PROGRAM general
VAR PERSISTENT
	//System date time function block
	system_date_time : date_time;
	//Daily reset bit, used throughout the program for any resets
	daily_reset : BOOL;
	//Alarm Acknoweldge unlatch timer
	alarm_ack_ton : ton;
	//Alarm Reset unlatch timer
	alarm_reset_ton : ton;
	//Alarm Ack and reset unlatch timer setpoint
	alarm_ack_unlatch_sp : TIME :=T#1S;
	
	//Always off bit
	always_off : BOOL := FALSE;
	
	//PLC States - move as needed
	ed_routine_idle : BOOL;
	ed_routine_cip : BOOL;
	ed_routine_manual : BOOL;
	ed_routine_maint : BOOL;
	ed_routine_stop : BOOL;
	ed_critical_stop : BOOL;
	
END_VAR

VAR
	//{attribute 'TcLinkTo' := 'TIID^Device 1 (EtherCAT)^Term 1 (EK1200)^Term 10 (EL2911)^StandardInputs^Standard Out Var 16'}
	twinsafe_safeout AT %I*: BOOL;
	
	//Linked manually
	twinsafe_status AT %I*: USINT;
	twinsafe_reset AT %Q*: BOOL;
	twinsafe_ack AT %Q*: BOOL;
	twinsafe_run AT %Q*: BOOL := TRUE;
	
	test_valve_position AT %I*: INT;
	
	
	test_valve: analog_scaling;
	test_nv_3110_a_open: BOOL;
	safety_reset_ton: TON;
END_VAR
VAR // added by the converter: edge detectors and wires of the graphical bodies
    _rt1, _rt2, _rt3, _rt4, _rt5 : R_TRIG;
    _w1, _w2, _w3, _w4 : BOOL;
END_VAR

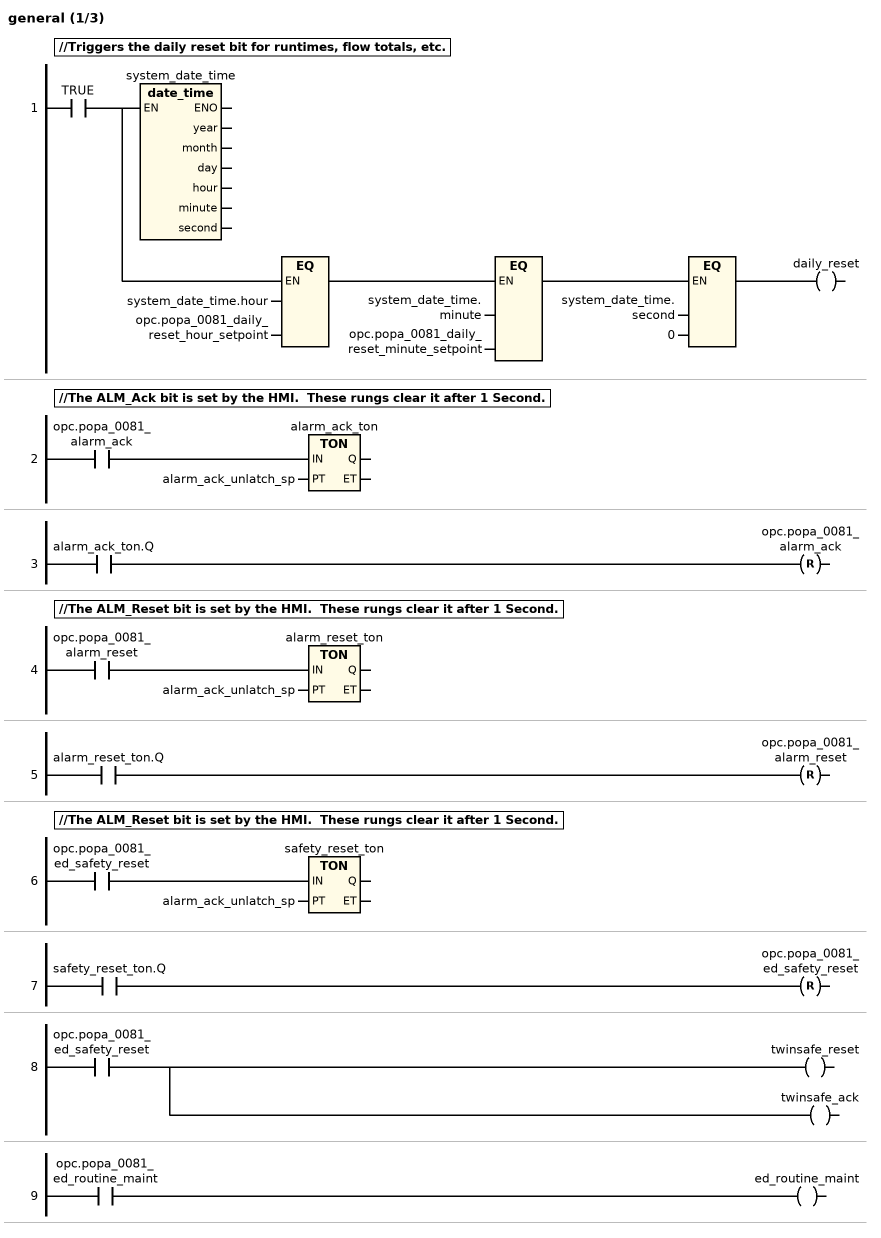
// NETWORK 1
// label: //Triggers the daily reset bit for runtimes, flow totals, etc.
system_date_time(); // date_time
daily_reset := system_date_time.hour = opc.popa_0081_daily_reset_hour_setpoint AND system_date_time.minute = opc.popa_0081_daily_reset_minute_setpoint AND system_date_time.second = 0;

// NETWORK 2
// label: //The ALM_Ack bit is set by the HMI.  These rungs clear it after 1 Second.
alarm_ack_ton(IN := opc.popa_0081_alarm_ack, PT := alarm_ack_unlatch_sp); // TON

// NETWORK 3
opc.popa_0081_alarm_ack R= alarm_ack_ton.Q;

// NETWORK 4
// label: //The ALM_Reset bit is set by the HMI.  These rungs clear it after 1 Second.
alarm_reset_ton(IN := opc.popa_0081_alarm_reset, PT := alarm_ack_unlatch_sp); // TON

// NETWORK 5
opc.popa_0081_alarm_reset R= alarm_reset_ton.Q;

// NETWORK 6
// label: //The ALM_Reset bit is set by the HMI.  These rungs clear it after 1 Second.
safety_reset_ton(IN := opc.popa_0081_ed_safety_reset, PT := alarm_ack_unlatch_sp); // TON

// NETWORK 7
opc.popa_0081_ed_safety_reset R= safety_reset_ton.Q;

// NETWORK 8
twinsafe_reset := opc.popa_0081_ed_safety_reset;
twinsafe_ack := opc.popa_0081_ed_safety_reset;

// NETWORK 9
ed_routine_maint := opc.popa_0081_ed_routine_maint;

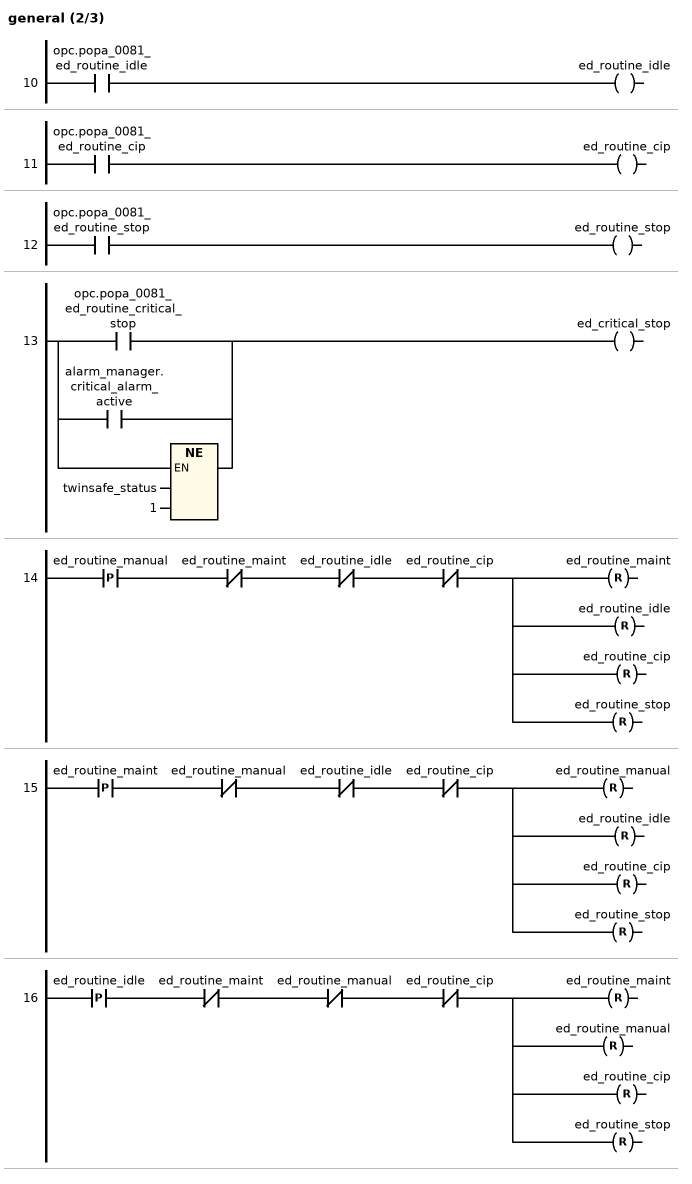
// NETWORK 10
ed_routine_idle := opc.popa_0081_ed_routine_idle;

// NETWORK 11
ed_routine_cip := opc.popa_0081_ed_routine_cip;

// NETWORK 12
ed_routine_stop := opc.popa_0081_ed_routine_stop;

// NETWORK 13
ed_critical_stop := opc.popa_0081_ed_routine_critical_stop OR alarm_manager.critical_alarm_active OR twinsafe_status <> 1;

// NETWORK 14
_rt1(CLK := ed_routine_manual);
_w1 := _rt1.Q AND NOT ed_routine_maint AND NOT ed_routine_idle AND NOT ed_routine_cip;
ed_routine_maint R= _w1;
ed_routine_idle R= _w1;
ed_routine_cip R= _w1;
ed_routine_stop R= _w1;

// NETWORK 15
_rt2(CLK := ed_routine_maint);
_w2 := _rt2.Q AND NOT ed_routine_manual AND NOT ed_routine_idle AND NOT ed_routine_cip;
ed_routine_manual R= _w2;
ed_routine_idle R= _w2;
ed_routine_cip R= _w2;
ed_routine_stop R= _w2;

// NETWORK 16
_rt3(CLK := ed_routine_idle);
_w3 := _rt3.Q AND NOT ed_routine_maint AND NOT ed_routine_manual AND NOT ed_routine_cip;
ed_routine_maint R= _w3;
ed_routine_manual R= _w3;
ed_routine_cip R= _w3;
ed_routine_stop R= _w3;

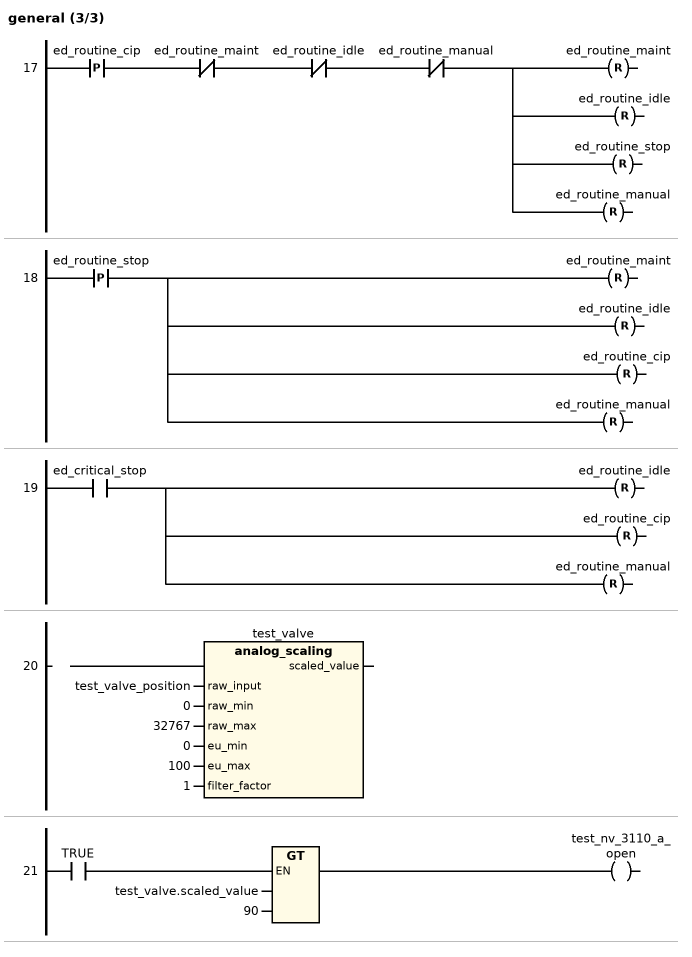
// NETWORK 17
_rt4(CLK := ed_routine_cip);
_w4 := _rt4.Q AND NOT ed_routine_maint AND NOT ed_routine_idle AND NOT ed_routine_manual;
ed_routine_maint R= _w4;
ed_routine_idle R= _w4;
ed_routine_stop R= _w4;
ed_routine_manual R= _w4;

// NETWORK 18
_rt5(CLK := ed_routine_stop);
ed_routine_maint R= _rt5.Q;
ed_routine_idle R= _rt5.Q;
ed_routine_cip R= _rt5.Q;
ed_routine_manual R= _rt5.Q;

// NETWORK 19
ed_routine_idle R= ed_critical_stop;
ed_routine_cip R= ed_critical_stop;
ed_routine_manual R= ed_critical_stop;

// NETWORK 20
test_valve(
    raw_input := test_valve_position,
    raw_min := 0,
    raw_max := 32767,
    eu_min := 0,
    eu_max := 100,
    filter_factor := 1); // analog_scaling

// NETWORK 21
test_nv_3110_a_open := test_valve.scaled_value > 90;

END_PROGRAM

(* stored: Version 1.1.0.1, ProductVersion 3.1.4024.15
   POU general: Id {afd5554c-a122-45cd-a612-91df6056dfdf}, SpecialFunc None *)
